FUNCTION_BLOCK FlushingSelector (* Basic Function Block Type *)
  (* Standard: 61499-2 *)
  (* Version 0.0, 6/22/2026, Schneider Electric, Template *)
  PACKAGE SE.Nereda;
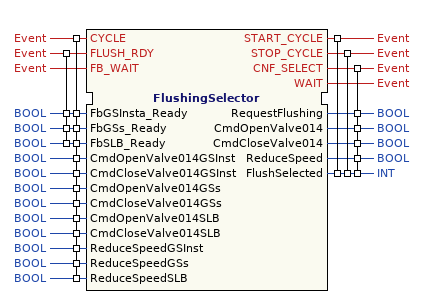
  EVENT_INPUT
    CYCLE WITH FbGSInsta_Ready, FbGSs_Ready, FbSLB_Ready, CmdOpenValve014GSInst, CmdCloseValve014GSInst, CmdOpenValve014GSs, CmdCloseValve014GSs, CmdOpenValve014SLB, CmdCloseValve014SLB, ReduceSpeedGSInst, ReduceSpeedGSs, ReduceSpeedSLB;
    FLUSH_RDY WITH FbGSInsta_Ready, FbGSs_Ready, FbSLB_Ready;
    FB_WAIT;
  END_EVENT
  EVENT_OUTPUT
    START_CYCLE WITH FlushSelected; (* Execution Confirmation *)
    STOP_CYCLE WITH FlushSelected;
    CNF_SELECT WITH RequestFlushing, CmdOpenValve014, CmdCloseValve014, FlushSelected, ReduceSpeed;
    WAIT;
  END_EVENT
  VAR_INPUT
    FbGSInsta_Ready : BOOL;
    FbGSs_Ready : BOOL;
    FbSLB_Ready : BOOL;
    CmdOpenValve014GSInst : BOOL;
    CmdCloseValve014GSInst : BOOL;
    CmdOpenValve014GSs : BOOL;
    CmdCloseValve014GSs : BOOL;
    CmdOpenValve014SLB : BOOL;
    CmdCloseValve014SLB : BOOL;
    ReduceSpeedGSInst : BOOL;
    ReduceSpeedGSs : BOOL;
    ReduceSpeedSLB : BOOL;
  END_VAR
  VAR_OUTPUT
    RequestFlushing : BOOL;
    CmdOpenValve014 : BOOL;
    CmdCloseValve014 : BOOL;
    ReduceSpeed : BOOL;
    FlushSelected : INT;
  END_VAR
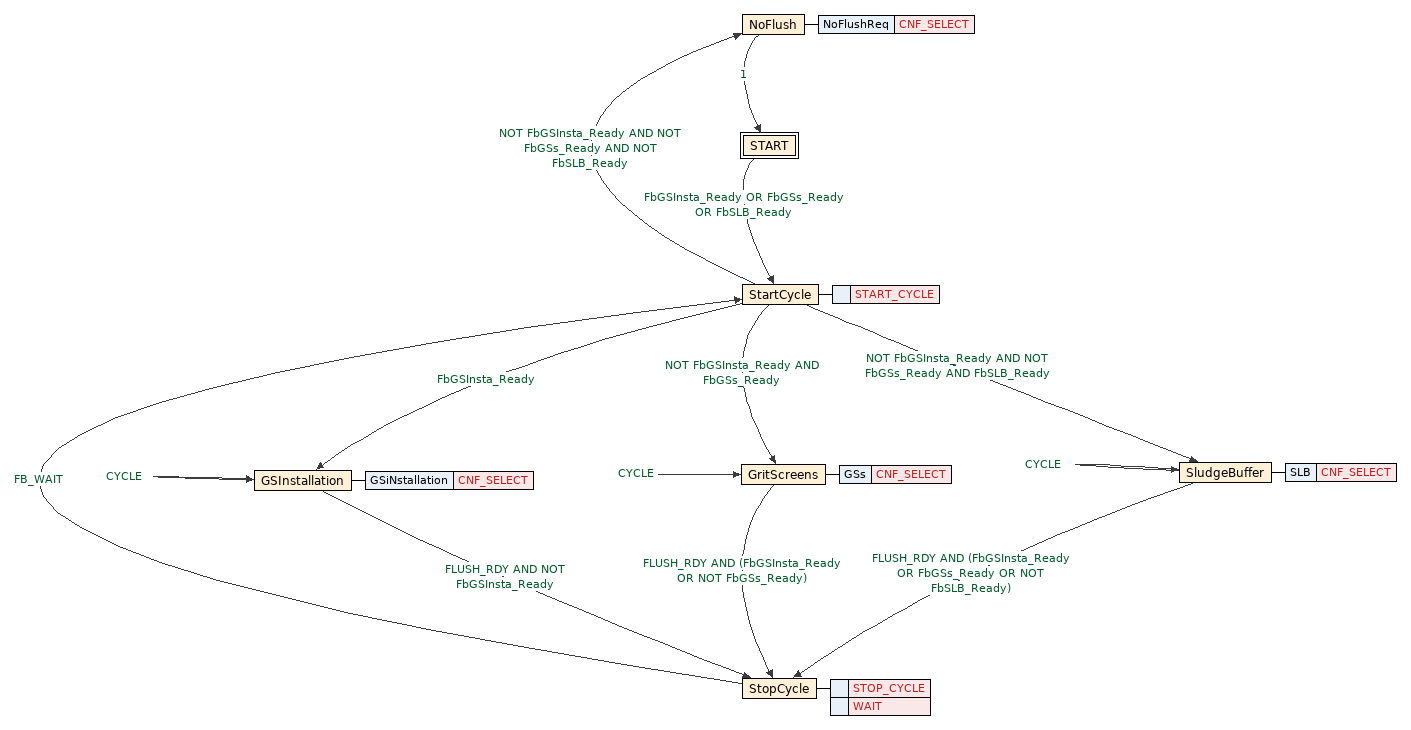
  EC_STATES
    START; (* Initial State *)
    GSInstallation : GSiNstallation -> CNF_SELECT;
    GritScreens : GSs -> CNF_SELECT;
    SludgeBuffer : SLB -> CNF_SELECT;
    StartCycle : -> START_CYCLE;
    StopCycle : -> STOP_CYCLE, -> WAIT;
    NoFlush : NoFlushReq -> CNF_SELECT;
  END_STATES
  EC_TRANSITIONS
    StartCycle TO GSInstallation := FbGSInsta_Ready;
    StartCycle TO GritScreens := NOT FbGSInsta_Ready AND FbGSs_Ready;
    StartCycle TO SludgeBuffer := NOT FbGSInsta_Ready AND NOT FbGSs_Ready AND FbSLB_Ready;
    START TO StartCycle := FbGSInsta_Ready OR FbGSs_Ready OR FbSLB_Ready;
    GSInstallation TO GSInstallation := CYCLE;
    GritScreens TO GritScreens := CYCLE;
    SludgeBuffer TO SludgeBuffer := CYCLE;
    SludgeBuffer TO StopCycle := FLUSH_RDY AND (FbGSInsta_Ready OR FbGSs_Ready OR NOT FbSLB_Ready);
    GritScreens TO StopCycle := FLUSH_RDY AND (FbGSInsta_Ready OR NOT FbGSs_Ready);
    GSInstallation TO StopCycle := FLUSH_RDY AND NOT FbGSInsta_Ready;
    StopCycle TO StartCycle := FB_WAIT;
    StartCycle TO NoFlush := NOT FbGSInsta_Ready AND NOT FbGSs_Ready AND NOT FbSLB_Ready;
    NoFlush TO START := 1;
  END_TRANSITIONS
  ALGORITHM GSiNstallation IN ST:
;
RequestFlushing := TRUE;
CmdOpenValve014 := CmdOpenValve014GSInst;
CmdCloseValve014 := CmdCloseValve014GSInst;
ReduceSpeed := ReduceSpeedGSInst;
FlushSelected := 1;
  END_ALGORITHM
  ALGORITHM GSs IN ST:
;
RequestFlushing := TRUE;
CmdOpenValve014 := CmdOpenValve014GSs;
CmdCloseValve014 := CmdCloseValve014GSs;
ReduceSpeed := ReduceSpeedGSs;
FlushSelected := 2;
  END_ALGORITHM
  ALGORITHM SLB IN ST:
;
RequestFlushing := TRUE;
CmdOpenValve014 := CmdOpenValve014SLB;
CmdCloseValve014 := CmdCloseValve014SLB;
ReduceSpeed := ReduceSpeedSLB;
FlushSelected := 3;
  END_ALGORITHM
  ALGORITHM NoFlushReq IN ST:
;
RequestFlushing := FALSE;
CmdOpenValve014 := TRUE;
CmdCloseValve014 := FALSE;
ReduceSpeed := FALSE;
FlushSelected := 0;
  END_ALGORITHM
END_FUNCTION_BLOCK
